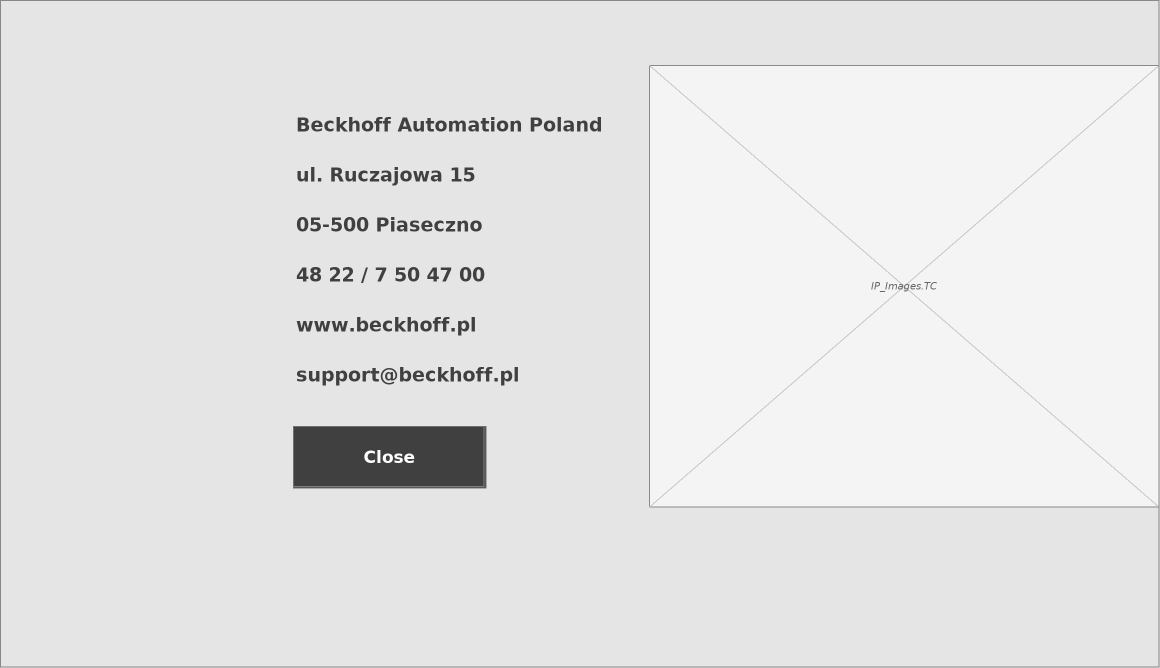
VISUALIZATION V_Home  // 1160x668
VAR_IN_OUT
	bKillProcess							: BOOL;
	sImageOsName							: STRING(20);
END_VAR
    Label (293,100 360x50), "Beckhoff Automation Poland"
    Label (293,150 360x50), "ul. Ruczajowa 15"
    Label (293,200 360x50), "05-500 Piaseczno"
    Label (293,250 360x50), "48 22 / 7 50 47 00"
    Label (293,300 360x50), "www.beckhoff.pl"
    Label (293,350 360x50), "support@beckhoff.pl"
    Image (649,65 510x442), image: IP_Images.TC
    Button (293,426 193x62), "Close", invisible if: sImageOsName='Windows CE'
        tap bKillProcess
END_VISUALIZATION

(* stored: Version 1.1.0.1, ProductVersion 3.1.4024.3
   Visu V_Home: Id {5e8e92e7-59ee-411f-b047-166382e2392a} *)
